# EPICS autosave request: pico8App/Db/pico8_settings.req
$(P)$(R)NumPoints

file "NDArrayBase_settings.req", P=$(P), R=$(R)
